// TIA Portal V18 export
TYPE "TD_Modes"
   STRUCT
      Drill : Int;
      DrillReverse : Int := 1;
      MUSpin : Int := 2;
      MUTorque : Int := 3;
      BO : Int := 4;
      Oscillate : Int := 5;
      Bypass : Int := 6;
   END_STRUCT;
END_TYPE
